// TIA Portal V17 export
// export: Created 2023-12-22T15:08:09.7897339Z, ExportSetting WithDefaults, DisplayName Totally Integrated Automation Portal, DisplayVersion V17, DisplayName TIA Portal Openness, DisplayVersion V17, DisplayName TIA Portal Version Control Interface, DisplayVersion V17, DisplayName STEP 7 Professional, DisplayVersion V17, DisplayName STEP 7 Safety, DisplayVersion V17, DisplayName WinCC Advanced, DisplayVersion V17
DATA_BLOCK "PE_Diag_DB"   // DB2
VERSION : 0.1
// stored: AutoNumber false, DBAccessibleFromOPCUA true, DBAccessibleFromWebserver true, InstanceOfName PE_Diag, InstanceOfType FB
"PE_Diag"
   // VAR_INPUT
   //    PE_1 : Real;
   //    PE_2 : Real;
   // END_VAR
   // VAR_OUTPUT
   //    PE : Real;
   // END_VAR
   // VAR
   //    Select : Bool;
   //    Delta : Real;
   //    Delta_In : Real;
   //    Delta_Max { S7_SetPoint := 'True'} : Real := 0.05;
   //    Warning : Word;
   // END_VAR
BEGIN
END_DATA_BLOCK
